FUNCTION_BLOCK ChipboardEx EXTENDS SectionEx
VAR_IN_OUT
	A21_SC_C18 : ConveyorSC;
	A21_LSC_C19 : ConveyorLSC;
	A21_LSC_C20 : ConveyorLSC;
END_VAR
VAR_IN_OUT
	robotLeft, robotRight : RobotA21;
	toolStorageLeft, toolStorageRight : A21ToolStorage;
	
	skidLeft, skidRight : SkidMagazine;
END_VAR
VAR	
	step : (IDLE, RETRACT_CONVEYOR, LOAD_CIP, EXTEND_CONVEYOR, COMPLETE := 1050);
	
	loadSet : INT;
END_VAR
VAR //bundle data
	materialsArr : (*REFERENCE TO*) ARRAY[0..CONSTS.maxPairs] OF PositionMaterials;
END_VAR
VAR
	aoiLoadLeft, aoiLoadRight : AOI_LoadChipboard;
	
	pushSmallConveyorPos : REAL;
	pushLargeConveyorPos : REAL;
END_VAR

aoiBlocks(); //call AOIs and large library FBs

SUPER^();

METHOD PROTECTED aoiBlocks : BOOL
VAR_INPUT
END_VAR
{warning disable C0371}
aoiLoadRight(
	sectionID:= sectionID, 
	execute:= ,
	robot:= robotRight, 
	storage:= skidRight,
	loadedMaterials:= loadedMaterials,
	surfaceID:= , 
	material:= , 
	loadedMaterials=> , 
	done=> , 
	error=> );
	
aoiLoadRight(
	sectionID:= sectionID, 
	execute:= , 
	robot:= robotRight, 
	storage:= skidRight,
	loadedMaterials:= loadedMaterials, 
	surfaceID:= , 
	material:= , 
	busy=> , 
	done=> , 
	error=> , 
	recovery=> , 
	failCounter=> );
END_METHOD

METHOD PROTECTED load : BOOL
VAR_INPUT
	pairIndex : INT;
END_VAR
VAR_OUTPUT
	error : BOOL;
END_VAR
VAR
	pair : REFERENCE TO PositionMaterials REF= materialsArr[pairIndex];
END_VAR
{warning disable C0371}
IF robotLeft.error AND robotLeft.error THEN
	error := TRUE;
	RETURN;

ELSIF
	( robotLeft.reservation <> sectionID AND_THEN robotLeft.reserve(sectionID) ) OR
	( robotRight.reservation <> sectionID AND_THEN robotRight.reserve(sectionID) ) THEN
	RETURN;
	
ELSIF //wrong tool and not finished changing tool
	(robotLeft.tool <> sectionID AND_THEN NOT robotLeft.changeEOAT(targetTool := sectionID)) OR
	(robotRight.tool <> sectionID AND_THEN NOT robotRight.changeEOAT(targetTool := sectionID))
THEN
	RETURN;
END_IF
//robots ok

CASE loadSet OF
	0: //left robot -> top, right robot -> bottom
		IF aoiLoadLeft.done AND aoiLoadRight.done THEN
			aoiLoadLeft.execute := aoiLoadRight.execute := FALSE;
			loadSet := 10;
			RETURN;
		END_IF
		
		aoiLoadLeft.surfaceID := Surface.TOP;
		aoiLoadLeft.material := pair.left;
		
		aoiLoadRight.surfaceID := Surface.BOTTOM;
		aoiLoadRight.material := pair.right;
		
		aoiLoadLeft.execute := NOT aoiLoadLeft.recovery;
		aoiLoadRight.execute := NOT aoiLoadRight.recovery;
		
	10: //recovery		
		IF robotRight.error THEN //left ok, right error
			
			IF aoiLoadLeft.done THEN
				aoiLoadLeft.execute := FALSE;
				loadSet := COMPLETE;
				RETURN;
			END_IF
			
			aoiLoadLeft.surfaceID := Surface.BOTTOM;
			aoiLoadLeft.material := pair.bottom;
			aoiLoadLeft.execute := NOT aoiLoadLeft.recovery;
			
		ELSIF robotLeft.error THEN //left error, right ok
			
			IF aoiLoadRight.done THEN
				aoiLoadRight.execute := FALSE;
				loadSet := COMPLETE;
				RETURN;
			END_IF
			
			aoiLoadRight.surfaceID := Surface.TOP;
			aoiLoadRight.material := pair.top;
			aoiLoadRight.execute := NOT aoiLoadRight.recovery;
			
		END_IF
		
	COMPLETE:
		loadSet := 0;
		
		robotLeft.release(sectionID);
		robotRight.release(sectionID);
		
		load := TRUE;
END_CASE
END_METHOD

METHOD PRIVATE loadingSequence : BOOL
VAR_IN_OUT
	robot : RobotA21;
	storage : SkidMagazine;
	loadStep : INT;
END_VAR
VAR_INPUT
	surfaceID : Surface;
	material : STRING;
END_VAR
VAR_OUTPUT
	fail : BOOL;
END_VAR
VAR
	slot : INT;
END_VAR
VAR CONSTANT
	suctionDistance : INT := 10;
END_VAR
{warning disable C0371}
IF material = '' THEN
	loadingSequence := TRUE;
	RETURN;
END_IF

CASE loadStep OF
	0:
		robot.clearCommand();
		IF robot.Ready THEN
			loadStep := 1;
		END_IF
	
	1:
		IF surfaceID = Surface.BOTTOM (*AND_THEN conveyors not retracted*) THEN
			//retract conveyors
			RETURN;
		END_IF
		loadStep := 10;
		
	10: //grab from chipboard skid
		IF NOT storage.findSlot(material := material, index => slot) THEN
			fail := TRUE;
			RETURN;
		(*
		ELSIF surfaceID = Surface.BOTTOM (*AND_THEN (*conveyor not lowered*)*) THEN
			//lower conveyor
			RETURN;
		*)
		END_IF
		
		IF robot.eoatDistance < suctionDistance THEN
			robot.HoldMaterial := storage.getSlot(i := slot);
		END_IF
		
		IF robot.Done THEN
			loadStep := COMPLETE;
			RETURN;
		ELSIF robot.materialAtHoldingPosition.4 OR robot.materialAtHoldingPosition.5 THEN //bits 4 and 5 are chipboard in position
			loadStep := 20;
			RETURN;
		END_IF
		
		robot.setGroup(group := 1, value := TaskA21.PLACE_CHIPBOARD_TOP);
		robot.setGroup(group := 2, value := slot);
		
	20: //place to bundle
		IF robotLeft.Done THEN
			loadStep := COMPLETE;
			RETURN;
		END_IF
		
		IF robot.HoldMaterial <> '' THEN
			loadedMaterials[surfaceID] := robot.HoldMaterial;
			robot.HoldMaterial := '';
		END_IF
		
	COMPLETE:
		IF loadedMaterials[surfaceID] = material THEN
			loadingSequence := TRUE;
		ELSE
			loadStep := 0;
		END_IF
		
END_CASE
END_METHOD

METHOD PROTECTED maintenance : BOOL
VAR_INPUT
END_VAR
{warning disable C0371}
//no specific tasks yet, free run and testing

IF robotLeft.Done THEN
	robotLeft.clearCommand();
END_IF

IF robotRight.Done THEN
	robotRight.clearCommand();
END_IF
END_METHOD

METHOD PROTECTED manual : BOOL
VAR_INPUT
END_VAR
END_METHOD

METHOD PROTECTED process : BOOL
VAR_INPUT
	auto : BOOL;
END_VAR
VAR_OUTPUT
	error : BOOL;
END_VAR
CASE step OF
	IDLE:
		IF trigger.Q THEN
			step := RETRACT_CONVEYOR;
		END_IF
		
	RETRACT_CONVEYOR:
		(*
		IF demoPair.bottom <> '' (*retract conveyors*) THEN
			IF TRUE (*BLSC 1-3 retracted*) THEN
				done := TRUE;
			END_IF
		ELSE
			done := TRUE;
		END_IF
		
		IF
			(manualStep AND_THEN execute) OR
			(NOT manualStep AND_THEN done)
		THEN
			done := FALSE;
			step := LOAD_MATERIAL;
		END_IF
		*)
		step := LOAD_CIP;
	LOAD_CIP:
		IF NOT done THEN
			done := load(pairIndex:= iPair, error=> error);
		END_IF
		
		IF
			(auto AND done) OR
			(NOT auto AND_THEN trigger.Q)
		THEN
			done := FALSE;
			
			step := EXTEND_CONVEYOR;
		END_IF
		
	EXTEND_CONVEYOR:
		(*
		IF FALSE (*conveyors not extended*) THEN
			//extend conveyors
		END_IF
		
		IF
			(auto AND done) OR
			(NOT auto AND_THEN execute) //conveyors extended
		THEN
			done := FALSE;
			step := COMPLETE;
		END_IF
		*)
		step := COMPLETE;
	COMPLETE:
		//reset everything
		step := IDLE;
		
		process := TRUE;
		
END_CASE
END_METHOD

METHOD PROTECTED ps_AbortCondition : BOOL
VAR_INPUT
END_VAR
{warning disable C0371}
ps_AbortCondition :=
	robotLeft.error OR 
	robotRight.error;
END_METHOD

METHOD PROTECTED ps_Aborted : BOOL
VAR_INPUT
END_VAR
ps_Aborted := TRUE;
END_METHOD

METHOD PROTECTED ps_Aborting : BOOL
VAR_INPUT
END_VAR
{warning disable C0371}
aoiLoadLeft.reset();
aoiLoadRight.reset();

robotLeft.clearCommand();
robotRight.clearCommand();

//stop conveyors

ps_Aborting :=
	NOT robotLeft.Busy AND
	NOT robotRight.Busy;
END_METHOD

METHOD PROTECTED ps_Clearing : BOOL
VAR_INPUT
END_VAR
{warning disable C0371}
(*reset conveyors*)

ps_Clearing := 
	NOT robotLeft.error AND
	NOT robotRight.error;
END_METHOD

METHOD PROTECTED ps_Complete : BOOL
VAR_INPUT
END_VAR
ps_Complete := TRUE;
END_METHOD

METHOD PROTECTED ps_Completing : BOOL
VAR_INPUT
END_VAR
ps_Completing := NOT occupied;
END_METHOD

METHOD PROTECTED ps_Held : BOOL
VAR_INPUT
END_VAR
ps_Held := NOT hold;
END_METHOD

METHOD PROTECTED ps_HoldCondition : BOOL
VAR_INPUT
END_VAR
END_METHOD

METHOD PROTECTED ps_Holding : BOOL
VAR_INPUT
END_VAR
{warning disable C0371}
//set robot to pause

ps_Holding := TRUE;
END_METHOD

METHOD PROTECTED ps_Resetting : BOOL
VAR_INPUT
END_VAR
{warning disable C0371}
(*reset conveyors*)

ps_Resetting := 
	reset AND
	NOT robotLeft.error AND
	NOT robotRight.error;
END_METHOD

METHOD PROTECTED ps_Starting : BOOL
VAR_INPUT
END_VAR
{warning disable C0371}
//extend conveyors

ps_Starting := TRUE; //conveyors extended
END_METHOD

METHOD PROTECTED ps_StopCondition : BOOL
VAR_INPUT
END_VAR
ps_StopCondition := 
	stop;
END_METHOD

METHOD PROTECTED ps_Stopped : BOOL
VAR_INPUT
END_VAR
ps_Stopped := TRUE;
END_METHOD

METHOD PROTECTED ps_Stopping : BOOL
VAR_INPUT
END_VAR
{warning disable C0371}
aoiLoadLeft.reset();
aoiLoadRight.reset();

robotLeft.clearCommand();
robotRight.clearCommand();

//stop conveyors

ps_Stopping :=
	NOT robotLeft.Busy AND
	NOT robotRight.Busy;
END_METHOD

METHOD PROTECTED ps_SuspendCondition : BOOL
VAR_INPUT
END_VAR
END_METHOD

METHOD PROTECTED ps_Suspended : BOOL
VAR_INPUT
END_VAR
ps_Suspended := NOT ps_SuspendCondition();
END_METHOD

METHOD PROTECTED ps_Suspending : BOOL
VAR_INPUT
END_VAR
ps_Suspending := TRUE;
END_METHOD

METHOD PROTECTED ps_Unholding : BOOL
VAR_INPUT
END_VAR
ps_Unholding := TRUE;
END_METHOD

METHOD PROTECTED ps_Unsuspending : BOOL
VAR_INPUT
END_VAR
ps_Unsuspending := TRUE;
END_METHOD

METHOD PROTECTED runSectionTasks : BOOL
VAR_INPUT
	auto : BOOL;
END_VAR
VAR_OUTPUT
	error : BOOL;
END_VAR
SUPER^.runSectionTasks(auto := auto, error => error);

CASE status OF //add additional instructions for each state
	SectionTask.IDLE:
		//
	
	SectionTask.ALIGN:
		//
		
	SectionTask.ACTIVE:
		//
		
	SectionTask.DISCHARGE:
		aoiLoadLeft.reset();
		aoiLoadRight.reset();
		
	SectionTask.COMPLETE:	
		//
		
	-100:
		RETURN;
		
END_CASE
END_METHOD

METHOD PROTECTED unload : BOOL
VAR_INPUT
END_VAR
//unload from insertion
//remove from staging table
END_METHOD

END_FUNCTION_BLOCK

(* stored: Version 1.1.0.1, ProductVersion 3.1.4024.11
   POU ChipboardEx: Id {4fb9c3b0-6386-4034-a58f-58f8ce2d611a}, SpecialFunc None
   Folder Actions_Cyclic: Id {1d4cf889-3e68-46d8-ad77-8ad472520e03}
   Folder PML Conditions: Id {db3fb587-f62c-413e-86fe-ffc9cd2d39ad}
   Folder PML Inter. States: Id {ab9cbcbe-212b-4c2d-a6dc-6cefed8dd476}
   Method aoiBlocks: Id {3aed7339-6bf5-4e31-a3ab-5532ab7d73f9}
   Method load: Id {fb843105-64e1-44e7-8bcd-619ab2de166a}
   Method loadingSequence: Id {96d77f50-a148-46c4-8ea5-43c584f562c9}
   Method maintenance: Id {8ea8cc70-de6a-428d-95f1-128be1ff5518}
   Method manual: Id {49a04b51-5215-4de4-bc90-fa8fd41f9b96}
   Method process: Id {4451bc85-ba29-4c10-8925-9cecf5fa2b5d}
   Method ps_AbortCondition: Id {a4e02a6f-1dd9-4b5b-975e-f31a9e1a9d39}
   Method ps_Aborted: Id {afdc7db0-3b5b-4aee-9866-560224678255}
   Method ps_Aborting: Id {bcb80c20-bb9a-4602-aac8-f5e829bea7b5}
   Method ps_Clearing: Id {b2125dae-b934-401c-82c0-ec5c61aac454}
   Method ps_Complete: Id {3a58560f-0a59-46c9-bc57-3f927e6c5604}
   Method ps_Completing: Id {ae85e936-b28f-40b1-88cf-bf1e6568a8fb}
   Method ps_Held: Id {5d3a9043-e079-4b24-8274-400f24d0d74b}
   Method ps_HoldCondition: Id {41e2994c-5099-4940-b7c7-3e4fc759762f}
   Method ps_Holding: Id {643ec6b6-c148-4c47-8dc1-33bcf2229aa8}
   Method ps_Resetting: Id {983ac4dd-1ff6-4e0c-b73e-4225e8740385}
   Method ps_Starting: Id {2f649bf5-415a-4c25-bab7-838c2c091e48}
   Method ps_StopCondition: Id {407cd14f-28d7-4012-b3c5-757c8224f570}
   Method ps_Stopped: Id {aa28d534-a613-452a-b2e0-8f44d37a695f}
   Method ps_Stopping: Id {9f68947d-2675-4ef1-bbb2-5fc51830c320}
   Method ps_SuspendCondition: Id {8bba2239-2ad5-48af-8103-232f2ea190d9}
   Method ps_Suspended: Id {a84b5a2d-37b2-4437-9dbc-913b7d65499c}
   Method ps_Suspending: Id {f12d78f3-9e13-4f1a-976e-cd31dc68bfd8}
   Method ps_Unholding: Id {3da58b83-15b5-4a80-962d-24acd5d42995}
   Method ps_Unsuspending: Id {e2a4d5ca-b527-4c8d-89e6-c12afb3c8b6c}
   Method runSectionTasks: Id {69ae0f9c-3b7e-4f7d-9514-05a650ec0734}
   Method unload: Id {f6db5e74-df8c-4b7a-9a29-336483c6ebce} *)
